{attribute 'pack_mode' := '2'}
TYPE ST_NC_PARAMETER :
STRUCT
  ParameterNumber : Tc2_MC2.MC_AxisParameter;
  rValue          : LREAL; // value (Bools are cast to real)
END_STRUCT
END_TYPE

(* stored: Version 1.1.0.1, ProductVersion 3.1.4024.12
   DUT ST_NC_PARAMETER: Id {d8fa3fa9-5e1a-0e1a-20db-dde782faeec2} *)
